// TIA Portal V15.1 export
// export: Created 2024-06-21T08:40:53.2574836Z, ExportSetting WithDefaults, DisplayName Totally Integrated Automation Portal, DisplayVersion V15.1 Update 5, DisplayName TIA Portal Openness, DisplayVersion V15.1 Update 5, DisplayName SINAMICS Startdrive Advanced, DisplayVersion V15.1, DisplayName G130, G150, S120, S150, SINAMICS MV, S210, DisplayVersion V15.1, DisplayName G110M, G120, G120C, G120D, G120P, DisplayVersion V15.1, DisplayName STEP 7 Professional, DisplayVersion V15.1 Update 5, DisplayName STEP 7 Safety, DisplayVersion V15.1, DisplayName WinCC Professional, DisplayVersion V15.1 Update 5, DisplayName SIMATIC Visualization Architect, DisplayVersion V15.1
FUNCTION_BLOCK "LPulse"   // FB1013, FBD
TITLE = LPulse
{ S7_Optimized_Access := 'FALSE' }
AUTHOR : VCC
FAMILY : Control
NAME : TimerON
VERSION : 1.0
// ================================================================================
// LPulse is used when a delay is necessary without using timer from Siemens.
// This timer has 2 ways to run:
// * Input = true constantly and pulse output 
// 
// Timer reset when input = false
// Timer reset when input reset = true 
// 
// For each case, Timer is reset when O_TimerValue >= I_MaxTimerValue
// ================================================================================
// stored: AutoNumber false, IsIECCheckEnabled false, SetENOAutomatically False, UDAEnableTagReadback false
   VAR_INPUT
      I_StartTimer { ExternalAccessible := 'False'; ExternalVisible := 'False'; ExternalWritable := 'False'} : Bool;   // Start Timer
      I_ResetTimer { ExternalAccessible := 'False'; ExternalVisible := 'False'; ExternalWritable := 'False'} : Bool;   // ResetTimer when I_MemstartTimer active
      I_MaxTimerValue { ExternalAccessible := 'False'; ExternalVisible := 'False'; ExternalWritable := 'False'} : DInt;   // Maximum Timer Value (1 unit = 1ms and max=7FFFFFFF)
   END_VAR
   VAR_OUTPUT
      O_TimerResult { ExternalAccessible := 'False'; ExternalVisible := 'False'; ExternalWritable := 'False'} : Bool;   // Timer result when time = MaxTime
      O_TimerValue { ExternalAccessible := 'False'; ExternalVisible := 'False'; ExternalWritable := 'False'} : DInt;   // Current timer value
   END_VAR
   VAR DB_SPECIFIC
      PulseStart { ExternalAccessible := 'False'; ExternalVisible := 'False'; ExternalWritable := 'False'} : Bool;   // Positive Pulse Start Timer
      MemStartTimer { ExternalAccessible := 'False'; ExternalVisible := 'False'; ExternalWritable := 'False'} : Bool;   // Memory of start timer
      PulseMemStart { ExternalAccessible := 'False'; ExternalVisible := 'False'; ExternalWritable := 'False'} : Bool;   // Positive Pulse Memory Start Timer
      StartTimeValue { ExternalAccessible := 'False'; ExternalVisible := 'False'; ExternalWritable := 'False'} : DInt;   // Start time value
      RunningTimeValue { ExternalAccessible := 'False'; ExternalVisible := 'False'; ExternalWritable := 'False'} : DInt;   // Running time value
      ElapsedTimeValue { ExternalAccessible := 'False'; ExternalVisible := 'False'; ExternalWritable := 'False'} : DInt;   // elapsed time value
   END_VAR
   VAR_TEMP
      T_Int : DInt;   // Temporally value
   END_VAR
   VAR_TEMP   // added for the SCL form of the ladder/FBD networks
      _w1 : Bool;
   END_VAR
BEGIN

REGION Network 1: **** 4.4 - Machine Status - Calculated **** Timer is running
   // Timer is running
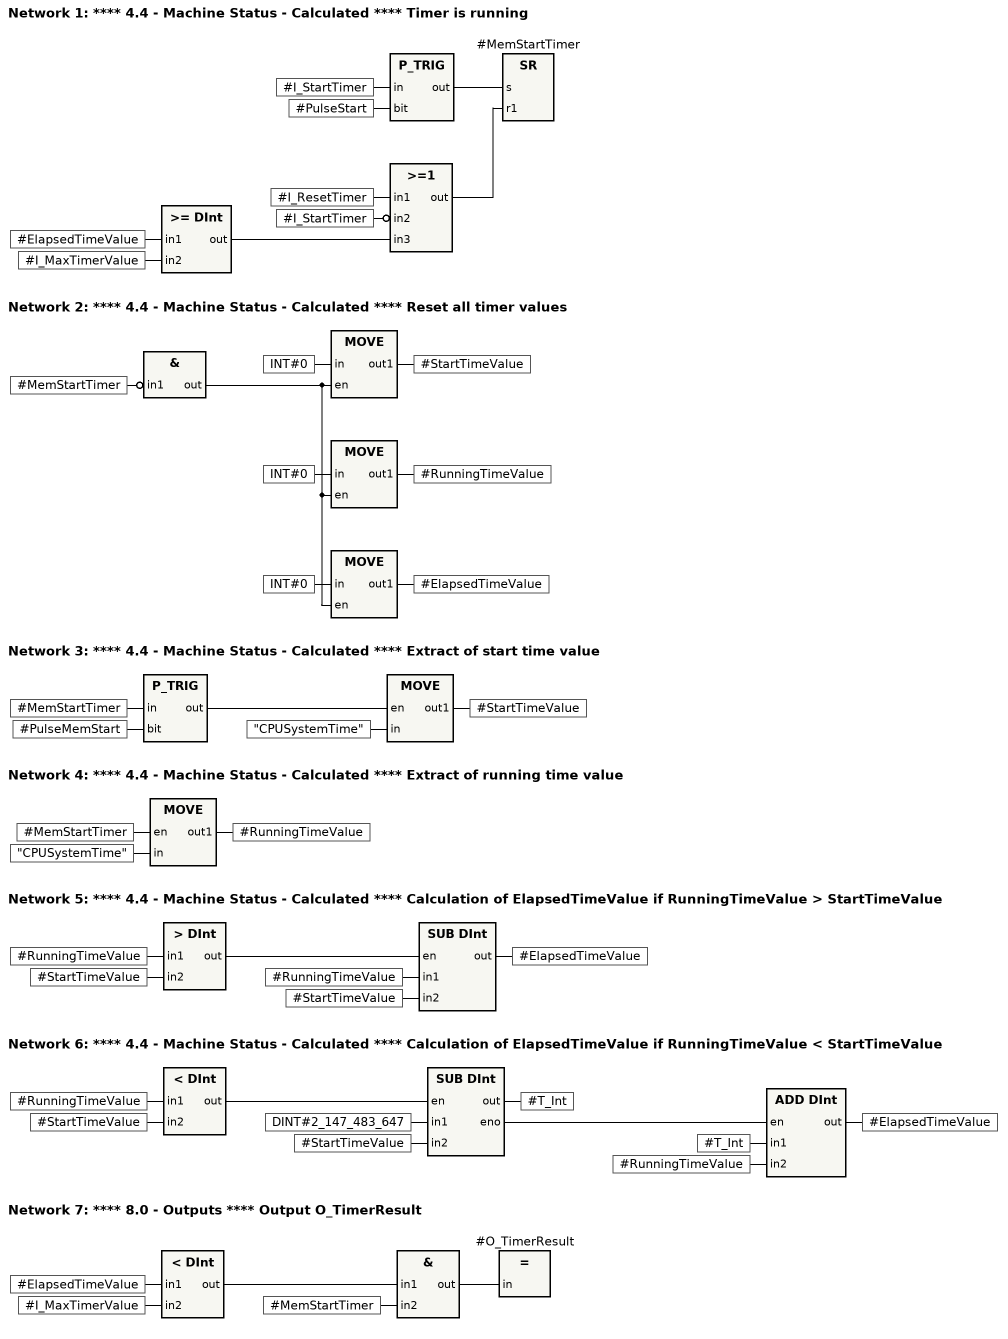
   #_w1 := #I_StartTimer AND NOT #PulseStart;   // rising edge
   #PulseStart := #I_StartTimer;
   IF #_w1 THEN
       #MemStartTimer := TRUE;   // SR flip-flop
   END_IF;
   IF #I_ResetTimer OR NOT #I_StartTimer OR (#ElapsedTimeValue >= #I_MaxTimerValue) THEN
       #MemStartTimer := FALSE;
   END_IF;
END_REGION

REGION Network 2: **** 4.4 - Machine Status - Calculated **** Reset all timer values
   // Reset all timer values
   IF NOT #MemStartTimer THEN
       #StartTimeValue := INT#0;
       #RunningTimeValue := INT#0;
       #ElapsedTimeValue := INT#0;
   END_IF;
END_REGION

REGION Network 3: **** 4.4 - Machine Status - Calculated **** Extract of start time value
   // Extract of start time value
   #_w1 := #MemStartTimer AND NOT #PulseMemStart;   // rising edge
   #PulseMemStart := #MemStartTimer;
   IF #_w1 THEN #StartTimeValue := "CPUSystemTime"; END_IF;
END_REGION

REGION Network 4: **** 4.4 - Machine Status - Calculated **** Extract of running time value
   // Extract of running time value
   IF #MemStartTimer THEN #RunningTimeValue := "CPUSystemTime"; END_IF;
END_REGION

REGION Network 5: **** 4.4 - Machine Status - Calculated **** Calculation of ElapsedTimeValue if RunningTimeValue > StartTimeValue
   // Calculation of ElapsedTimeValue if RunningTimeValue > StartTimeValue
   IF #RunningTimeValue > #StartTimeValue THEN
       #ElapsedTimeValue := #RunningTimeValue - #StartTimeValue;
   END_IF;
END_REGION

REGION Network 6: **** 4.4 - Machine Status - Calculated **** Calculation of ElapsedTimeValue if RunningTimeValue < StartTimeValue
   // Calculation of ElapsedTimeValue if RunningTimeValue < StartTimeValue
   // ENO of a box is taken as its EN; it also drops when the box reports an error
   IF #RunningTimeValue < #StartTimeValue THEN
       #T_Int := DINT#2_147_483_647 - #StartTimeValue;
       #ElapsedTimeValue := #T_Int + #RunningTimeValue;
   END_IF;
END_REGION

REGION Network 7: **** 8.0 - Outputs **** Output O_TimerResult
   // Output O_TimerResult
   #O_TimerResult := (#ElapsedTimeValue < #I_MaxTimerValue) AND #MemStartTimer;
END_REGION

REGION Network 8: **** 8.0 - Outputs **** Copy of TimerValue to output O_TimerValue
   // Copy of TimerValue to output O_TimerValue
   // Copy of HoldValue to output O_HoldValue
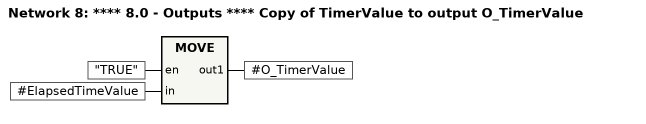
   IF "TRUE" THEN #O_TimerValue := #ElapsedTimeValue; END_IF;
END_REGION
END_FUNCTION_BLOCK
